{attribute 'qualified_only'}
VAR_GLOBAL
	stData	:data;
END_VAR

(* stored: Version 1.1.0.1, ProductVersion 3.1.4024.12
   GVL GVL: Id {8a525c67-4920-4136-bf9a-29393a240c19} *)
